// TIA Portal V16 export
// export: Created 2022-02-04T14:40:28.4923421Z, ExportSetting WithDefaults, DisplayName Totally Integrated Automation Portal, DisplayVersion V16 Update 1, DisplayName TIA Portal Version Control Interface, DisplayVersion V16, DisplayName TIA Portal Openness, DisplayVersion V16, DisplayName SINAMICS Startdrive Advanced, DisplayVersion V16 Update 5, DisplayName SINAMICS Startdrive G130, G150, S120, S150, SINAMICS MV, S210, DisplayVersion V16 Update 5, DisplayName SINAMICS Startdrive G110M, G120, G120C, G120D, G120P, G115D, DisplayVersion V16 Update 5, DisplayName STEP 7 Professional, DisplayVersion V16, DisplayName STEP 7 Safety, DisplayVersion V16, DisplayName WinCC Advanced, DisplayVersion V16, DisplayName SIMATIC Visualization Architect, DisplayVersion V16
TYPE "PlankOnChain"
// stored: IsFailsafeCompliant false
   STRUCT
      Chain : Bool;   // Цепь, на которйо ледит доска (0 - низкая, 1 - высокая)
      NoEmpty : Bool;   // есть доска на цепи
      Length : Int;   // Длина уложенной доски
   END_STRUCT;
END_TYPE
